// this interface is only necessary to allow type-checking for Value Expressions
INTERFACE IValExp EXTENDS __System.IQueryInterface

END_INTERFACE

(* stored: Version 1.1.0.1, ProductVersion 3.1.4024.12
   Itf IValExp: Id {e141454d-c68e-40e9-a30d-1af90c8c8770} *)
